// TIA Portal V18 export
// export: Created 2026-01-09T11:31:56.5978943Z, ExportSetting WithDefaults, DisplayName Totally Integrated Automation Portal, DisplayVersion V18 Update 5, DisplayName TIA Portal Openness, DisplayVersion V18 Update 5, DisplayName TIA Portal Teamcenter Gateway, DisplayVersion V18, DisplayName TIA Portal Version Control Interface, DisplayVersion V18, DisplayName SINAMICS Startdrive Advanced, DisplayVersion V18 SP2 Update 1, DisplayName SINAMICS Startdrive G110M, G120, G120C, G120D, G120P, G115D, DisplayVersion V18 SP2 Update 1, DisplayName SINAMICS Startdrive G130, G150, S120, S150, SINAMICS MV, S210, G220, S200, DisplayVersion V18 SP2 Update 1, DisplayName STEP 7 Professional, DisplayVersion V18 Update 5, DisplayName STEP 7 Safety, DisplayVersion V18, DisplayName WinCC Professional, DisplayVersion V18 Update 5
TagTable "ToolingCode"
  AutoProcessData.A_Table1_Code1 : String  (PLC tag AutoProcessData.A_Table_1[1].Code, CPU S71500-2PN_TP700, 1 s)
  AutoProcessData.A_Table1_Code2 : String  (PLC tag AutoProcessData.A_Table_1[2].Code, CPU S71500-2PN_TP700, 1 s)
  AutoProcessData.A_Table1_Code3 : String  (PLC tag AutoProcessData.A_Table_1[3].Code, CPU S71500-2PN_TP700, 1 s)
  AutoProcessData.A_Table1_Code4 : String  (PLC tag AutoProcessData.A_Table_1[4].Code, CPU S71500-2PN_TP700, 1 s)
  AutoProcessData.A_Table1_Code5 : String  (PLC tag AutoProcessData.A_Table_1[5].Code, CPU S71500-2PN_TP700, 1 s)
  AutoProcessData.A_Table1_Code6 : String  (PLC tag AutoProcessData.A_Table_1[6].Code, CPU S71500-2PN_TP700, 1 s)
  AutoProcessData.A_Table1_Code7 : String  (PLC tag AutoProcessData.A_Table_1[7].Code, CPU S71500-2PN_TP700, 1 s)
  AutoProcessData.A_Table1_Code8 : String  (PLC tag AutoProcessData.A_Table_1[8].Code, CPU S71500-2PN_TP700, 1 s)
  AutoProcessData.A_Table2_Code1 : String  (PLC tag AutoProcessData.A_Table_2[1].Code, CPU S71500-2PN_TP700, 1 s)
  AutoProcessData.A_Table2_Code2 : String  (PLC tag AutoProcessData.A_Table_2[2].Code, CPU S71500-2PN_TP700, 1 s)
  AutoProcessData.A_Table2_Code3 : String  (PLC tag AutoProcessData.A_Table_2[3].Code, CPU S71500-2PN_TP700, 1 s)
  AutoProcessData.A_Table2_Code4 : String  (PLC tag AutoProcessData.A_Table_2[4].Code, CPU S71500-2PN_TP700, 1 s)
  AutoProcessData.A_Table2_Code5 : String  (PLC tag AutoProcessData.A_Table_2[5].Code, CPU S71500-2PN_TP700, 1 s)
  AutoProcessData.A_Table2_Code6 : String  (PLC tag AutoProcessData.A_Table_2[6].Code, CPU S71500-2PN_TP700, 1 s)
  AutoProcessData.A_Table2_Code7 : String  (PLC tag AutoProcessData.A_Table_2[7].Code, CPU S71500-2PN_TP700, 1 s)
  AutoProcessData.A_Table2_Code8 : String  (PLC tag AutoProcessData.A_Table_2[8].Code, CPU S71500-2PN_TP700, 1 s)
  AutoProcessData.FixtureCode_A1_1 : String  (PLC tag AutoProcessData.FixtureCode_A1[1], CPU S71500-2PN_TP700, 1 s)
  AutoProcessData.FixtureCode_A1_2 : String  (PLC tag AutoProcessData.FixtureCode_A1[2], CPU S71500-2PN_TP700, 1 s)
  AutoProcessData.FixtureCode_A1_3 : String  (PLC tag AutoProcessData.FixtureCode_A1[3], CPU S71500-2PN_TP700, 1 s)
  AutoProcessData.FixtureCode_A1_4 : String  (PLC tag AutoProcessData.FixtureCode_A1[4], CPU S71500-2PN_TP700, 1 s)
  AutoProcessData.FixtureCode_A1_5 : String  (PLC tag AutoProcessData.FixtureCode_A1[5], CPU S71500-2PN_TP700, 1 s)
  AutoProcessData.FixtureCode_A2_1 : String  (PLC tag AutoProcessData.FixtureCode_A2[1], CPU S71500-2PN_TP700, 1 s)
  AutoProcessData.FixtureCode_A2_2 : String  (PLC tag AutoProcessData.FixtureCode_A2[2], CPU S71500-2PN_TP700, 1 s)
  AutoProcessData.FixtureCode_A2_3 : String  (PLC tag AutoProcessData.FixtureCode_A2[3], CPU S71500-2PN_TP700, 1 s)
  AutoProcessData.FixtureCode_A2_4 : String  (PLC tag AutoProcessData.FixtureCode_A2[4], CPU S71500-2PN_TP700, 1 s)
  AutoProcessData.FixtureCode_A2_5 : String  (PLC tag AutoProcessData.FixtureCode_A2[5], CPU S71500-2PN_TP700, 1 s)
  AutoProcessData.FixtureCode_A1_6 : String  (PLC tag AutoProcessData.FixtureCode_A1[6], CPU S71500-2PN_TP700, 1 s)
  AutoProcessData.FixtureCode_A1_7 : String  (PLC tag AutoProcessData.FixtureCode_A1[7], CPU S71500-2PN_TP700, 1 s)
  AutoProcessData.FixtureCode_A2_6 : String  (PLC tag AutoProcessData.FixtureCode_A2[6], CPU S71500-2PN_TP700, 1 s)
  AutoProcessData.FixtureCode_A2_7 : String  (PLC tag AutoProcessData.FixtureCode_A2[7], CPU S71500-2PN_TP700, 1 s)
  AutoProcessData.FixtureCode_A2_8 : String  (PLC tag AutoProcessData.FixtureCode_A2[8], CPU S71500-2PN_TP700, 1 s)
  AutoProcessData.GripperCode_R1[1] : String  (PLC tag AutoProcessData.GripperCode_R1[1], CPU S71500-2PN_TP700, 1 s)
  AutoProcessData.GripperCode_R1[2] : String  (PLC tag AutoProcessData.GripperCode_R1[2], CPU S71500-2PN_TP700, 1 s)
  AutoProcessData.GripperCode_R1[3] : String  (PLC tag AutoProcessData.GripperCode_R1[3], CPU S71500-2PN_TP700, 1 s)
  AutoProcessData.GripperCode_R1[4] : String  (PLC tag AutoProcessData.GripperCode_R1[4], CPU S71500-2PN_TP700, 1 s)
  AutoProcessData.GripperCode_R2[1] : String  (PLC tag AutoProcessData.GripperCode_R2[1], CPU S71500-2PN_TP700, 1 s)
  AutoProcessData.GripperCode_R2[2] : String  (PLC tag AutoProcessData.GripperCode_R2[2], CPU S71500-2PN_TP700, 1 s)
  AutoProcessData.GripperCode_R2[3] : String  (PLC tag AutoProcessData.GripperCode_R2[3], CPU S71500-2PN_TP700, 1 s)
  AutoProcessData.GripperCode_R2[4] : String  (PLC tag AutoProcessData.GripperCode_R2[4], CPU S71500-2PN_TP700, 1 s)
  AutoProcessData.GripperCode_R3[1] : String  (PLC tag AutoProcessData.GripperCode_R3[1], CPU S71500-2PN_TP700, 1 s)
  AutoProcessData.GripperCode_R3[2] : String  (PLC tag AutoProcessData.GripperCode_R3[2], CPU S71500-2PN_TP700, 1 s)
  AutoProcessData.GripperCode_R3[3] : String  (PLC tag AutoProcessData.GripperCode_R3[3], CPU S71500-2PN_TP700, 1 s)
  AutoProcessData.GripperCode_R3[4] : String  (PLC tag AutoProcessData.GripperCode_R3[4], CPU S71500-2PN_TP700, 1 s)
